// TIA Portal V21 export
TYPE "motorHMI"
   STRUCT
      status : Word;
      "step" : USInt;
      stepTime : LTime;
      speedSp : Real;
      speedPv : Real;
      alm { S7_SetPoint := 'True'} : Word;
      stopCtx { S7_SetPoint := 'True'} : "stopCtxHMI";
   END_STRUCT;
END_TYPE
